SUBAPPLICATION Seitenschieber (* Subapplication Type *)
  (* Standard: 61499-2 *)
  (* Version 1.0, 2023-01-29, Franz *)
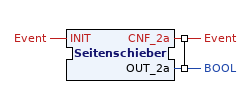
  EVENT_INPUT
    INIT;
  END_EVENT
  EVENT_OUTPUT
    CNF_2a WITH OUT_2a;
  END_EVENT
  VAR_OUTPUT
    OUT_2a : BOOL;
  END_VAR
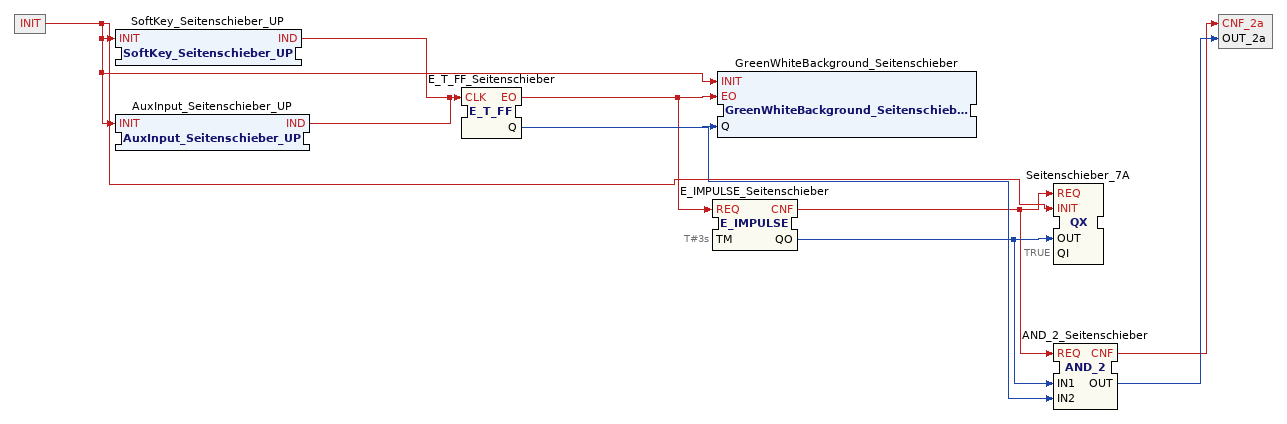
  FBS
    AND_2_Seitenschieber : AND_2;
    E_T_FF_Seitenschieber : E_T_FF;
    Seitenschieber_7A : QX(QI := TRUE);
    E_IMPULSE_Seitenschieber : E_IMPULSE(TM := T#3s);
  END_FBS
  SUBAPPS
    GreenWhiteBackground_Seitenschieber : GreenWhiteBackground_Seitenschieber;
    AuxInput_Seitenschieber_UP : AuxInput_Seitenschieber_UP;
    SoftKey_Seitenschieber_UP : SoftKey_Seitenschieber_UP;
  END_SUBAPPS
  EVENT_CONNECTIONS
    E_IMPULSE_Seitenschieber.CNF TO AND_2_Seitenschieber.REQ;
    E_T_FF_Seitenschieber.EO TO E_IMPULSE_Seitenschieber.REQ;
    E_IMPULSE_Seitenschieber.CNF TO Seitenschieber_7A.REQ;
    AND_2_Seitenschieber.CNF TO CNF_2a;
    INIT TO Seitenschieber_7A.INIT;
    INIT TO GreenWhiteBackground_Seitenschieber.INIT;
    E_T_FF_Seitenschieber.EO TO GreenWhiteBackground_Seitenschieber.EO;
    INIT TO AuxInput_Seitenschieber_UP.INIT;
    AuxInput_Seitenschieber_UP.IND TO E_T_FF_Seitenschieber.CLK;
    INIT TO SoftKey_Seitenschieber_UP.INIT;
    SoftKey_Seitenschieber_UP.IND TO E_T_FF_Seitenschieber.CLK;
  END_CONNECTIONS
  DATA_CONNECTIONS
    E_IMPULSE_Seitenschieber.QO TO AND_2_Seitenschieber.IN1;
    E_T_FF_Seitenschieber.Q TO AND_2_Seitenschieber.IN2; (* Schieber offen *)
    E_IMPULSE_Seitenschieber.QO TO Seitenschieber_7A.OUT;
    AND_2_Seitenschieber.OUT TO OUT_2a;
    E_T_FF_Seitenschieber.Q TO GreenWhiteBackground_Seitenschieber.Q; (* Schieber offen *)
  END_CONNECTIONS
END_SUBAPPLICATION
